FUNCTION_BLOCK FB_SimCell
VAR_INPUT
END_VAR
VAR_OUTPUT
END_VAR
VAR
	bPartPresentAtInfeed		AT %Q* : BOOL;
	bPartPresentAtOutfeed		AT %Q* : BOOL;
	
	fbInfeedActuator			: FB_SimActuator;
	fbOutfeedActuator			: FB_SimActuator;
	fbInfeedConveyor			: FB_SimAxis;
	fbOutfeedConveyor			: FB_SimAxis;
	fbIndexConveyor				: FB_SimAxis;
	
	fbSimScanner				: FB_SimBarcodeScanner;
	fbSimFiller					: FB_SimFiller;
	fbSimCapper					: FB_SimCapper;
	fbSimWeigher				: FB_SimCheckWeigher;
	
	fbTmr						: ARRAY[0..9] OF TON;
	rand						: ARRAY[0..9] OF DRAND;
	i,j,k						: INT;
	bStationLoaded				: ARRAY[0..3] OF BOOL;
	
	iIndexState					: DINT;
	iInfeedState				: DINT;
END_VAR

FOR i := 0 TO 9 DO
	rand[i](Seed:=i);
END_FOR

fbInfeedActuator();
fbInfeedConveyor();
fbIndexConveyor();
fbOutfeedActuator();
fbOutfeedConveyor();

fbSimScanner();
fbSimFiller();
fbSimCapper();
fbSimWeigher();

// Infeed
CASE iInfeedState OF
	0:
		fbTmr[0].PT := TO_TIME(1000 + rand[0].Num * 1000);
		iInfeedState := 1;
		
	1:
		fbTmr[0](IN:=(fbInfeedConveyor.State <> 0 AND NOT bPartPresentAtInfeed));
		IF fbTmr[0].Q THEN
			fbTmr[0](IN:=FALSE);
			bPartPresentAtInfeed := TRUE;
			iInfeedState := 2;
		END_IF
		
	2:
		IF fbInfeedActuator.bExtended THEN
			bPartPresentAtInfeed := FALSE;
			fbSimScanner.PartPresent := TRUE;
			bStationLoaded[0] := TRUE;
			iInfeedState := 3;
		END_IF
	
	3:
		iInfeedState := 0;
		
END_CASE


CASE iIndexState OF
	0:
		// conveyor indexing
		IF fbIndexConveyor.bMoveAbsCmd AND 
			(fbIndexConveyor.fActPosition <> fbIndexConveyor.fPositionCmd) THEN
			iIndexState := 1;
		END_IF
		
	1:
		fbSimScanner.PartPresent := FALSE;
		fbSimFiller.PartPresent := FALSE;
		fbSimCapper.PartPresent := FALSE;
		fbSimWeigher.PartPresent := FALSE;
		
		// index complete
		IF fbIndexConveyor.fActPosition = fbIndexConveyor.fPositionCmd THEN
			iIndexState := 2;
		END_IF
		
	2:
		// shift parts
		fbSimScanner.PartPresent := FALSE;
		fbSimFiller.PartPresent := bStationLoaded[0];
		fbSimCapper.PartPresent := bStationLoaded[1];
		fbSimWeigher.PartPresent := bStationLoaded[2];
		
		bStationLoaded[3] := bStationLoaded[2];
		bStationLoaded[2] := bStationLoaded[1];
		bStationLoaded[1] := bStationLoaded[0];
		bStationLoaded[0] := FALSE;
		
		iIndexState := 0;
		
END_CASE

END_FUNCTION_BLOCK

(* stored: Version 1.1.0.1, ProductVersion 3.1.4024.12
   POU FB_SimCell: Id {04fe6bf7-e7cc-4102-8854-b7f2cb31d082}, SpecialFunc None *)
